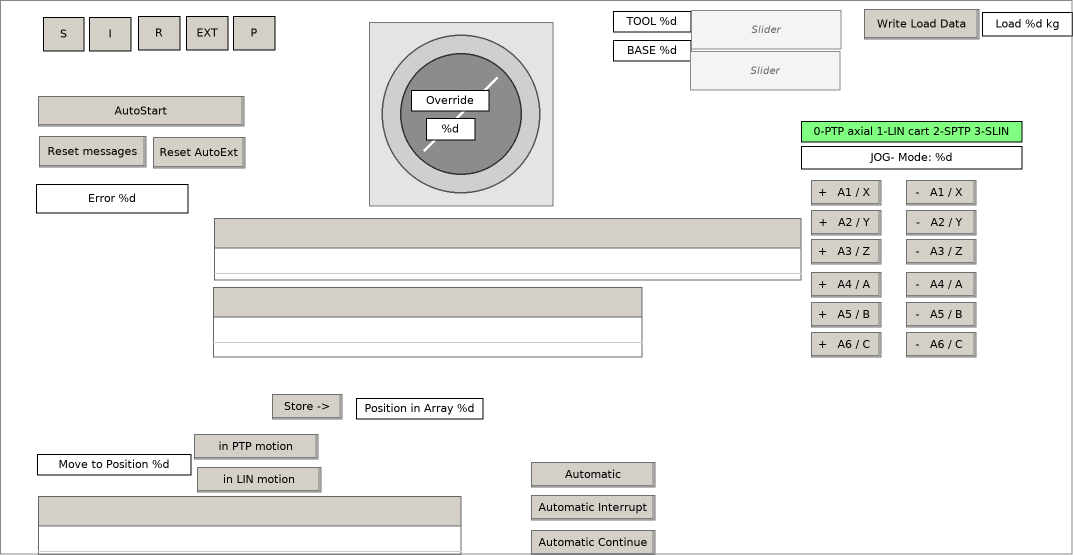
VISUALIZATION HMI_dmeo  // 1073x555
    Potentiometer360 (362,22 198x184), variable: GVL.nOverrideGlobal, style: Potentiometer-Potentiometer360-Gray, scale format: %d, scale 0..100
    Rectangle (411,90 78x21), "Override"
    Rectangle (426,118 49x22), "%d", text variable: GVL.nOverrideGlobal
        OnMouseClick: write the text variable via VisuDialogs.Numpad
    Button (38,96 206x30), "AutoStart", colour toggle: MAIN.bAutostartDone
        tap GVL.HMI_AutoStart
    Button (39,136 107x31), "Reset messages"
        tap GVL.HMI_MessageReset
    Rectangle (613,11 78x21), "TOOL %d", text variable: GVL.HMI_TOOL
        OnMouseClick: write the text variable via Default, min 1, max 16
    Rectangle (613,40 78x21), "BASE %d", text variable: GVL.HMI_BASE
        OnMouseClick: write the text variable via Default, min 1, max 16
    Slider (691,10 150x39), variable: GVL.HMI_TOOL, scale 0..5
    Slider (690,51 150x39), variable: GVL.HMI_BASE, scale 0..5
    Line (808,124)
    Rectangle (801,146 221x23), "JOG- Mode: %d", text variable: mxA_Motion.nJogMoveType
        OnMouseClick: write the text variable via Default, min 0, max 3
    Button (811,180 70x25), "+ A1 / X"
        tap mxA_Motion.bJogA1_P
    Button (906,180 70x25), "- A1 / X"
        tap mxA_Motion.bJogA1_M
    Button (864,9 115x30), "Write Load Data"
        tap GVL.HMI_WriteLoadData
    Rectangle (982,12 91x24), "Load %d kg", text variable: GVL.HMI_LOAD
        OnMouseClick: write the text variable via Default
    Rectangle (801,121 221x21), "0-PTP axial 1-LIN cart 2-SPTP 3-SLIN"
    Button (811,210 70x25), "+ A2 / Y"
        tap mxA_Motion.bJogA2_P
    Button (906,210 70x25), "- A2 / Y"
        tap mxA_Motion.bJogA2_M
    Button (811,239 70x25), "+ A3 / Z"
        tap mxA_Motion.bJogA3_P
    Button (906,239 70x25), "- A3 / Z"
        tap mxA_Motion.bJogA3_M
    Button (811,272 70x25), "+ A4 / A"
        tap mxA_Motion.bJogA4_P
    Button (906,272 70x25), "- A4 / A"
        tap mxA_Motion.bJogA4_M
    Button (811,302 70x25), "+ A5 / B"
        tap mxA_Motion.bJogA5_P
    Button (906,302 70x25), "- A5 / B"
        tap mxA_Motion.bJogA5_M
    Button (811,332 70x25), "+ A6 / C"
        tap mxA_Motion.bJogA6_P
    Button (906,332 70x25), "- A6 / C"
        tap mxA_Motion.bJogA6_M
    Rectangle (43,17 41x34), "S", colour toggle: GVL.HMI_Error_SINT
    Rectangle (233,16 42x34), "P", colour toggle: GVL.HMI_Error_ProConOS
    Rectangle (89,17 42x34), "I", colour toggle: GVL.HMI_DrivesNotReady
    Rectangle (138,16 42x34), "R", colour toggle: MAIN.bAutostartDispActive
    Rectangle (186,16 42x34), "EXT", colour toggle: GVL.HMI_AutoEXT
    Rectangle (36,184 152x29), "Error %d", text variable: GVL.HMI_Error_General_ID, colour toggle: GVL.HMI_Error_General
    Table (214,218 587x62), data array: GVL.HMI_ActualCartPos
        p3854506369: GVL.HMI_ActualCartPos.X
        p1892666644: GVL.HMI_ActualCartPos.Y
        p338671338: GVL.HMI_ActualCartPos.Z
        p2170511999: GVL.HMI_ActualCartPos.A
        p3723444502: GVL.HMI_ActualCartPos.B
        p1218418051: GVL.HMI_ActualCartPos.C
        p746581629: GVL.HMI_ActualCartPos.Status
        p3104783080: GVL.HMI_ActualCartPos.Turn
        p2501879983: GVL.HMI_ActualCartPos.E1
        p7306298: GVL.HMI_ActualCartPos.E2
        p1933151965: GVL.HMI_ActualCartPos.E3
        p3863566920: GVL.HMI_ActualCartPos.E4
        p2192122294: GVL.HMI_ActualCartPos.E5
        p400160035: GVL.HMI_ActualCartPos.E6
    Table (213,287 429x70), data array: GVL.HMI_ActualAxisPosition
        p3854506369: GVL.HMI_ActualAxisPosition.A1
        p1892666644: GVL.HMI_ActualAxisPosition.A2
        p338671338: GVL.HMI_ActualAxisPosition.A3
        p2170511999: GVL.HMI_ActualAxisPosition.A4
        p3723444502: GVL.HMI_ActualAxisPosition.A5
        p1218418051: GVL.HMI_ActualAxisPosition.A6
        p746581629: GVL.HMI_ActualAxisPosition.E1
        p3104783080: GVL.HMI_ActualAxisPosition.E2
        p2501879983: GVL.HMI_ActualAxisPosition.E3
        p7306298: GVL.HMI_ActualAxisPosition.E4
        p1933151965: GVL.HMI_ActualAxisPosition.E5
        p3863566920: GVL.HMI_ActualAxisPosition.E6
        p2192122294: ActualKarthPositon.E5
        p400160035: ActualKarthPositon.E6
    Button (153,137 92x31), "Reset AutoExt"
        tap MAIN.bAutoExternReset
    Rectangle (356,398 127x21), "Position in Array %d", text variable: GVL.HMI_TouchUpIndex
        OnMouseClick: write the text variable via Default, min 1, max 100
    Button (272,394 70x25), "Store ->"
        tap GVL.HMI_TouchUpStoreNow
    Rectangle (37,454 154x21), "Move to Position %d", text variable: mxA_Motion.nMove_PositonMode_Pos
        OnMouseClick: write the text variable via Default, min 1, max 16
    Button (197,467 124x25), "in LIN motion"
        tap mxA_Motion.bMoveLinar_PositonMode
    Table (38,496 423x59), data array: GVL.aPosArray[mxA_Motion.nMove_PositonMode_Pos].E6AXIS
        p2192122294: ActualKarthPositon.E5
        p400160035: ActualKarthPositon.E6
        p3854506369: GVL.aPosArray[mxA_Motion.nMove_PositonMode_Pos].E6AXIS.A1
        p1892666644: GVL.aPosArray[mxA_Motion.nMove_PositonMode_Pos].E6AXIS.A2
        p338671338: GVL.aPosArray[mxA_Motion.nMove_PositonMode_Pos].E6AXIS.A3
        p2170511999: GVL.aPosArray[mxA_Motion.nMove_PositonMode_Pos].E6AXIS.A4
        p3723444502: GVL.aPosArray[mxA_Motion.nMove_PositonMode_Pos].E6AXIS.A5
        p1218418051: GVL.aPosArray[mxA_Motion.nMove_PositonMode_Pos].E6AXIS.A6
        p746581629: GVL.aPosArray[mxA_Motion.nMove_PositonMode_Pos].E6AXIS.E1
        p3104783080: GVL.aPosArray[mxA_Motion.nMove_PositonMode_Pos].E6AXIS.E2
        p2501879983: GVL.aPosArray[mxA_Motion.nMove_PositonMode_Pos].E6AXIS.E3
        p7306298: GVL.aPosArray[mxA_Motion.nMove_PositonMode_Pos].E6AXIS.E4
        p1933151965: GVL.aPosArray[mxA_Motion.nMove_PositonMode_Pos].E6AXIS.E5
        p3863566920: GVL.aPosArray[mxA_Motion.nMove_PositonMode_Pos].E6AXIS.E6
    Button (194,434 124x25), "in PTP motion"
        tap mxA_Motion.bMovePTP_PositonMode
    Button (531,462 124x25), "Automatic", colour toggle: mxA_Motion.bExecAutoDemo
        toggle mxA_Motion.bExecAutoDemo
    Button (531,495 124x25), "Automatic Interrupt"
        tap mxA_Motion.fbAutoDemo.fbKRC_Interrupt.Execute
    Button (531,530 124x25), "Automatic Continue"
        tap mxA_Motion.fbAutoDemo.fbKRC_Continue.Enable
END_VISUALIZATION

(* stored: Version 1.1.0.1, ProductVersion 3.1.4024.10
   Visu HMI_dmeo: Id {e45b569c-5b08-4b3a-afa6-6d9fce2872b4} *)
